FUNCTION_BLOCK FB_RollingAverage_Ppm
VAR CONSTANT
	LOW : UINT := 0;
	HIGH : UINT := 59;
END_VAR
VAR
	aCounts : ARRAY[LOW..HIGH] OF UINT;
	fbTimer : TON := (PT:=T#1S);
	nLatestIndex : UINT := LOW;
	bInitialized : BOOL;
	nIdx : UINT;
	bEnable : BOOL;
END_VAR

IF bEnable THEN
	fbTimer(IN := TRUE);
	IF fbTimer.Q THEN
		fbTimer(IN := FALSE);
		aCounts[nLatestIndex] := 0;
		nLatestIndex := (nLatestIndex + 1) MOD (HIGH + 1);
		IF (nLatestIndex = 0) THEN bInitialized := TRUE; END_IF
	END_IF
ELSE
	fbTimer(IN := FALSE);
	nLatestIndex := LOW;
	bInitialized := FALSE;
	FOR nIdx := LOW TO HIGH DO
		aCounts[nIdx] := 0;
	END_FOR
END_IF

{attribute 'monitoring' := 'call'}
PROPERTY Count : UINT
GET
Count := aCounts[nLatestIndex];
END_GET
END_PROPERTY

{attribute 'monitoring' := 'call'}
PROPERTY Enable : BOOL
GET
Enable := bEnable;
END_GET
SET
bEnable := Enable;
END_SET
END_PROPERTY

METHOD Increment
VAR
	nIdx : UINT;
END_VAR
FOR nIdx := LOW TO HIGH DO
	aCounts[nIdx] := aCounts[nIdx] + 1;
END_FOR
END_METHOD

{attribute 'monitoring' := 'call'}
PROPERTY Initialized : BOOL
GET
Initialized := bInitialized;
END_GET
END_PROPERTY

END_FUNCTION_BLOCK

(* stored: Version 1.1.0.1, ProductVersion 3.1.4024.12
   POU FB_RollingAverage_Ppm: Id {1f98aed1-8a87-4e4d-be94-2918753b949b}, SpecialFunc None
   Property Count: Id {267e785e-413b-4acd-b77f-09b0012f0c55}
   Get Get: Id {28fb3f5e-5c15-4ec0-b23b-e65b18489d7a}
   Property Enable: Id {02be5590-d706-419c-a92a-2f50b996aa52}
   Get Get: Id {86997190-cb15-461e-a742-5ffa1e119885}
   Set Set: Id {dd020c8e-2ed7-4535-b608-7ca40d880e47}
   Method Increment: Id {3f58cae1-0188-4a4b-8ca9-25da58294ef4}
   Property Initialized: Id {3f6b3dc1-3c6a-41be-b8ad-f706e8d555b3}
   Get Get: Id {095cc6d5-c49d-4b13-a933-88615a383b45} *)
